KUKA KRL program: MsgLib.src, MsgLib.dat

--- MsgLib.src ---
&ACCESS RV1
&REL 15
&COMMENT Message library
DEF MsgLib()
   ;**************************************************
   ;Creation Date: 7.12.2007
   ;Change:  23.06.2012 additional properties possible
   ;         for logging and advance stop control
   ;Change:  16.06.2023 modify MsgNotifyTextPar
   ;Change:  06.09.2023 modify MsgNotifyTextPar & zip code
   ;**************************************************
   ;FOLD Interfaces and message examples within this fold
      ;----------Global subroutines and functions: -------
      ;MsgNotify(sText[]:IN, sModul[]:IN, nNumPar:IN, sTextPar[]:IN, nMsgNr:IN,MsgOpt:IN)
      ;MsgNotifyTextPar(sText[]:IN, sModul[]:IN, nNumPar:IN, sTextPar[]:IN, sTextPar2[]:IN, nMsgNr:IN,MsgOpt:IN)
      ;MsgQuit(sText[]:IN, sModul[]:IN, nNumPar:IN, sTextPar[]:IN, nMsgNr:IN,MsgOpt:IN)
      ;MsgState(nHandle:OUT, sText[]:IN, sModul[]:IN, nNumPar:IN, sTextPar[]:IN, nMsgNr:IN,MsgOpt:IN)
      ;MsgLoop(sText[]:IN,sModul[]:IN)
      ;MsgDialog(nAnswer:OUT,sText[]:IN,sModul[]:IN,sTextPar[]:IN,sDialogSK1[]:IN,sDialogSK2[]:IN,sDialogSK3[]:IN,sDialogSK4[]:IN,sDialogSK5[]:IN,sDialogSK6[]:IN,sDialogSK7[]:IN,NoBrakes:IN, nMsgNr:IN,MsgOpt:IN)
      ;----------Explainations for parameters: -----------
      ;CHAR sText[]  message text or message DB-key (80 chars)
      ;CHAR sModul[] (option) modulname or key (24 char)
      ;INT nNumPar   (option)numeric value inserted in sText[] at the position %1
      ;CHAR sTextPar[] (option)text or message DB-key inserted in sText[] at the position %1 (26 char)
      ;MsgOpt          (option) Structure KrlMsgOpt_T  BOOL VL_Stop,Clear_P_Reset,Log_To_DB
      ;                (option) VL_Stop=TRUE    => Creates an advance stop | FALSE avoids this behavior
      ;                (option) Clear_P_Reset=TRUE (Default) deletes Messages at program reset / cancelled
      ;                (option) Log_To_DB=TRUE => entry into logbook => enfluence to system performance
      ;----------Examples: -------------------------------
      ;MsgNotifyTextPar("Error", "CrossMeld", 0, "Error message 1", "Error message 2", 511)
      ;MsgNotify("this is a notify message")
      ;MsgQuit("this is a quit message", "myMod")
      ;MsgQuit("this is a quit message", "myMod",,,12345)
      ;INT myInt=123
      ;MsgQuit("this is the %1 quit message", "Module", myInt)
      ;MsgNotify("this is a %1 notify message", "Tech", , "asd")
      ;MsgLoop("this is the loop message")
      ;MsgLoop(" "); cancels loop message
      ;MsgDialog(DialogAnswer, "DBKEY" OR "dialog message", "Module", "TextPar for %1 in DBKey", "DialogKey1", "DialogKey2", "DialogKey3",,,,,,12345)
      ;MsgDialog(DialogAnswer, "StartPTP", "CrossMeld", "Achse 3", "YES", "NO", "Cancel")
      ;MsgNotifyTextPar("DBKEY" OR "notify message", "Module", 0 OR >0, "TextPar for %1", "TextPar for %2")
      ;  nNumPar = 0: TextPar will be send as %1 %2
      ;  nNumPar <> 0: nNumPar will be send as %1
      ;  nNumPar = ,,: TextPar will be send as %1 %2
   ;ENDFOLD
END


GLOBAL DEF MsgNotify(sText[]:IN, sModul[]:IN, nNumPar:IN, sTextPar[]:IN, nMsgNr:IN, MsgOpt:IN)
   DECL CHAR sText[]
   DECL CHAR sModul[]
   DECL CHAR sTextPar[]
   DECL KrlMsg_T Msg
   DECL KrlMsgParType_T MsgParType
   DECL KrlMsgPar_T MsgPar[3]
   DECL KrlMsgOpt_T MsgOpt ;Bool-elements: VL_Stop,Clear_P_Reset,Log_To_DB
   DECL KrlMsgOpt_T DummyMsgOpt
   DECL State_T State
   DECL INT count, len, offset, nHandle
   DECL INT nNumPar
   DECL INT nMsgNr
   CheckOfMsgOpt(MsgOpt);Creates default values in case of none availability
   CheckOfMsgNr(Msg, nMsgNr);Creates default values in case of none availability
   CheckOfMsgText(Msg, sText[])
   CheckOfModulText(Msg, sModul[])
   ERR_CLEAR($ERR)
   ON_ERROR_PROCEED
   offset=nNumPar
   IF $ERR.Number == 0 THEN
      offset=0
      MsgPar[1].Par_Txt[]=" "
      Swrite(MsgPar[1].Par_Txt[], State, Offset, "%d", nNumPar)
      MsgPar[1].Par_type=#Value
   ELSE
      ERR_CLEAR($ERR)
      ON_ERROR_PROCEED
      len=STRLEN(sTextPar[])
      IF len > 0 THEN
         IF len > 26 THEN
            len=26
         ENDIF
         FOR count = 1 TO len
            MsgPar[1].Par_Txt[count]=sTextPar[count]
         ENDFOR
         MsgPar[1].Par_type=#Value
      ENDIF
   ENDIF
   nHandle=Set_KrlMsg(#NOTIFY, Msg, MsgPar[], MsgOpt)
END


GLOBAL DEF MsgQuit(sText[]:IN, sModul[]:IN, nNumPar:IN, sTextPar[]:IN, nMsgNr:IN, MsgOpt:IN)
   DECL CHAR sText[]
   DECL CHAR sModul[]
   DECL CHAR sTextPar[]
   DECL KrlMsg_T Msg
   DECL KrlMsgParType_T MsgParType
   DECL KrlMsgPar_T MsgPar[3]
   DECL KrlMsgOpt_T MsgOpt
   DECL KrlMsgOpt_T DummyMsgOpt
   DECL State_T State
   DECL INT count, len, offset, nHandle
   DECL INT nNumPar
   DECL INT nMsgNr
   CheckOfMsgOpt(MsgOpt);Creates default values in case of none availability
   CheckOfMsgNr(Msg, nMsgNr);Creates default values in case of none availability
   CheckOfMsgText(Msg, sText[])
   CheckOfModulText(Msg, sModul[])
   ERR_CLEAR($ERR)
   ON_ERROR_PROCEED
   offset=nNumPar
   IF $ERR.Number == 0 THEN
      offset=0
      MsgPar[1].Par_Txt[]=" "
      Swrite(MsgPar[1].Par_Txt[], State, offset, "%d", nNumPar)
      MsgPar[1].Par_type=#Value
   ELSE
      ERR_CLEAR($ERR)
      len=STRLEN(sTextPar[])
      IF len > 0 THEN
         IF len > 26 THEN
            len=26
         ENDIF
         FOR count = 1 TO len
            MsgPar[1].Par_Txt[count]=sTextPar[count]
         ENDFOR
         MsgPar[1].Par_type=#Value
      ENDIF
   ENDIF
   nHandle=Set_KrlMsg(#QUIT, Msg, MsgPar[], MsgOpt)
   WHILE (Exists_KrlMsg(nHandle))
      WAIT SEC 0.1
   ENDWHILE
END


GLOBAL DEF MsgState(nHandle:OUT, sText[]:IN, sModul[]:IN, nNumPar:IN, sTextPar[]:IN, nMsgNr:IN, MsgOpt:IN)
   DECL CHAR sText[]
   DECL CHAR sModul[]
   DECL CHAR sTextPar[]
   DECL KrlMsg_T Msg
   DECL KrlMsgParType_T MsgParType
   DECL KrlMsgPar_T MsgPar[3]
   DECL KrlMsgOpt_T MsgOpt
   DECL KrlMsgOpt_T DummyMsgOpt
   DECL State_T State
   DECL INT count, len, offset
   DECL INT nHandle
   DECL INT nNumPar
   DECL INT nMsgNr
   CheckOfMsgOpt(MsgOpt);Creates default values in case of none availability
   CheckOfMsgNr(Msg, nMsgNr);Creates default values in case of none availability
   CheckOfMsgText(Msg, sText[])
   CheckOfModulText(Msg, sModul[])
   ERR_CLEAR($ERR)
   ON_ERROR_PROCEED
   offset=nNumPar
   IF $ERR.Number == 0 THEN
      offset=0
      MsgPar[1].Par_Txt[]=" "
      Swrite(MsgPar[1].Par_Txt[], State, offset, "%d", nNumPar)
      MsgPar[1].Par_type=#Value
   ELSE
      ERR_CLEAR($ERR)
      len=STRLEN(sTextPar[])
      IF len > 0 THEN
         IF len > 26 THEN
            len=26
         ENDIF
         FOR count = 1 TO len
            MsgPar[1].Par_Txt[count]=sTextPar[count]
         ENDFOR
         MsgPar[1].Par_type=#Value
      ENDIF
   ENDIF
   nHandle=Set_KrlMsg(#STATE, Msg, MsgPar[], MsgOpt)
END


GLOBAL DEF MsgLoop(sText[]:IN, sModul[]:IN)
   DECL CHAR sText[]
   DECL CHAR sModul[]
   DECL CHAR sMsg[80]
   DECL CHAR sMod[24]
   DECL INT count, len
   len=STRLEN(sText[])
   IF len > 0 THEN
      IF len > 80 THEN
         len=80
      ENDIF
      FOR count = 1 TO len
         sMsg[count]=sText[count]
      ENDFOR
   ENDIF
   len=STRLEN(sModul[])
   IF len > 0 THEN
      IF len > 24 THEN
         len=24
      ENDIF
      FOR count = 1 TO len
         sMod[count]=sModul[count]
      ENDFOR
   ELSE
      sMod[]="Appl"
   ENDIF
   IF (STRLEN(sMsg[]) > 0) THEN
      IF lnHandle > 0 THEN
         WAIT FOR Clear_KrlMsg(lnHandle) OR TRUE
         lnHandle=0
      ENDIF
      FOR count = 1 TO STRLEN(sMsg[])
         IF sMsg[count] <> " " THEN
            MsgState(lnHandle, sMsg[], sMod[])
            EXIT
         ENDIF
      ENDFOR
   ENDIF
END


GLOBAL DEF MsgDialog(nAnswer:OUT, sText[]:IN, sModul[]:IN, sTextPar[]:IN, sDialogSK1[]:IN, sDialogSK2[]:IN, sDialogSK3[]:IN, sDialogSK4[]:IN, sDialogSK5[]:IN, sDialogSK6[]:IN, sDialogSK7[]:IN, NoBrakes:IN, nMsgNr:IN, MsgOpt:IN)
   DECL KrlMsg_T Msg
   DECL KrlMsgPar_T MsgPar[3]
   DECL KrlMsgOpt_T MsgOpt
   DECL KrlMsgOpt_T DummyMsgOpt
   DECL KrlMsgDlgSK_T Msg_SOFTKEY[7]
   DECL INT count, len, nHandle
   DECL INT nAnswer
   DECL INT nMsgNr
   DECL BOOL NoBrakes
   DECL CHAR sText[]
   DECL CHAR sModul[]
   DECL CHAR sTextPar[]
   DECL CHAR sDialogSK1[]
   DECL CHAR sDialogSK2[]
   DECL CHAR sDialogSK3[]
   DECL CHAR sDialogSK4[]
   DECL CHAR sDialogSK5[]
   DECL CHAR sDialogSK6[]
   DECL CHAR sDialogSK7[]
   DECL CHAR sMsg[80]
   CheckOfMsgOpt(MsgOpt);Creates default values in case of none availability
   CheckOfMsgNr(Msg, nMsgNr);Creates default values in case of none availability
   CheckOfMsgText(Msg, sText[])
   CheckOfModulText(Msg, sModul[])
   ERR_CLEAR($ERR)
   ON_ERROR_PROCEED
   len=STRLEN(sDialogSK1[])
   IF $ERR.Number == 0 THEN
      IF len > 0 THEN
         IF len > 24 THEN
            len=24
         ENDIF
         Msg_SOFTKEY[7].Sk_Type=#KEY
         FOR count = 1 TO len
            Msg_SOFTKEY[7].Sk_txt[count]=sDialogSK1[count]
         ENDFOR
      ENDIF
   ELSE
      FOR count = 1 TO 24
         Msg_SOFTKEY[7].Sk_txt[count]=" "
      ENDFOR
   ENDIF
   ERR_CLEAR($ERR)
   ON_ERROR_PROCEED
   len=STRLEN(sDialogSK2[])
   IF $ERR.Number == 0 THEN
      len=STRLEN(sDialogSK2[])
      IF len > 0 THEN
         IF len > 24 THEN
            len=24
         ENDIF
         Msg_SOFTKEY[6].Sk_Type=#KEY
         FOR count = 1 TO len
            Msg_SOFTKEY[6].Sk_txt[count]=sDialogSK2[count]
         ENDFOR
      ENDIF
   ELSE
      FOR count = 1 TO 24
         Msg_SOFTKEY[6].Sk_txt[count]=" "
      ENDFOR
   ENDIF
   ERR_CLEAR($ERR)
   ON_ERROR_PROCEED
   len=STRLEN(sDialogSK3[])
   IF $ERR.Number == 0 THEN
      len=STRLEN(sDialogSK3[])
      IF len > 0 THEN
         IF len > 24 THEN
            len=24
         ENDIF
         Msg_SOFTKEY[5].Sk_Type=#KEY
         FOR count = 1 TO len
            Msg_SOFTKEY[5].Sk_txt[count]=sDialogSK3[count]
         ENDFOR
      ENDIF
   ELSE
      FOR count = 1 TO 24
         Msg_SOFTKEY[5].Sk_txt[count]=" "
      ENDFOR
   ENDIF
   ERR_CLEAR($ERR)
   ON_ERROR_PROCEED
   len=STRLEN(sDialogSK4[])
   IF $ERR.Number == 0 THEN
      len=STRLEN(sDialogSK4[])
      IF len > 0 THEN
         IF len > 24 THEN
            len=24
         ENDIF
         Msg_SOFTKEY[4].Sk_Type=#KEY
         FOR count = 1 TO len
            Msg_SOFTKEY[4].Sk_txt[count]=sDialogSK4[count]
         ENDFOR
      ENDIF
   ELSE
      FOR count = 1 TO 24
         Msg_SOFTKEY[4].Sk_txt[count]=" "
      ENDFOR
   ENDIF
   ERR_CLEAR($ERR)
   ON_ERROR_PROCEED
   len=STRLEN(sDialogSK5[])
   IF $ERR.Number == 0 THEN
      len=STRLEN(sDialogSK5[])
      IF len > 0 THEN
         IF len > 24 THEN
            len=24
         ENDIF
         Msg_SOFTKEY[3].Sk_Type=#KEY
         FOR count = 1 TO len
            Msg_SOFTKEY[3].Sk_txt[count]=sDialogSK5[count]
         ENDFOR
      ENDIF
   ELSE
      FOR count = 1 TO 24
         Msg_SOFTKEY[3].Sk_txt[count]=" "
      ENDFOR
   ENDIF
   ERR_CLEAR($ERR)
   ON_ERROR_PROCEED
   len=STRLEN(sDialogSK6[])
   IF $ERR.Number == 0 THEN
      len=STRLEN(sDialogSK6[])
      IF len > 0 THEN
         IF len > 24 THEN
            len=24
         ENDIF
         Msg_SOFTKEY[2].Sk_Type=#KEY
         FOR count = 1 TO len
            Msg_SOFTKEY[2].Sk_txt[count]=sDialogSK6[count]
         ENDFOR
      ENDIF
   ELSE
      FOR count = 1 TO 24
         Msg_SOFTKEY[2].Sk_txt[count]=" "
      ENDFOR
   ENDIF
   ERR_CLEAR($ERR)
   ON_ERROR_PROCEED
   len=STRLEN(sDialogSK7[])
   IF $ERR.Number == 0 THEN
      len=STRLEN(sDialogSK7[])
      IF len > 0 THEN
         IF len > 24 THEN
            len=24
         ENDIF
         Msg_SOFTKEY[1].Sk_Type=#KEY
         FOR count = 1 TO len
            Msg_SOFTKEY[1].Sk_txt[count]=sDialogSK7[count]
         ENDFOR
      ENDIF
   ELSE
      FOR count = 1 TO 24
         Msg_SOFTKEY[1].Sk_txt[count]=" "
      ENDFOR
   ENDIF
   len=STRLEN(sTextPar[])
   IF len > 0 THEN
      IF len > 26 THEN
         len=26
      ENDIF
      FOR count = 1 TO len
         MsgPar[1].Par_Txt[count]=sTextPar[count]
      ENDFOR
      MsgPar[1].Par_type=#Value
   ENDIF
   nHandle=SET_KRLDLG(Msg, MsgPar[], Msg_SOFTKEY[], MsgOpt)
   ERR_CLEAR($ERR)
   ON_ERROR_PROCEED
   NoBrakes=NoBrakes
   IF NOT ($ERR.Number == 0) THEN
      NoBrakes=FALSE
   ENDIF
   IF (nHandle > 0) THEN
      WHILE (Exists_KrlDlg(nHandle, nAnswer))
         WAIT SEC 0.5
         IF NoBrakes THEN
            PTP $AXIS_ACT
         ENDIF
      ENDWHILE
   ENDIF
END


GLOBAL DEF MsgNotifyTextPar(sText[]:IN, sModul[]:IN, nNumPar:IN, sTextPar[]:IN, sTextPar2[]:IN, nMsgNr:IN, MsgOpt:IN)
   DECL CHAR sText[]
   DECL CHAR sModul[]
   DECL CHAR sTextPar[]
   DECL CHAR sTextPar2[]
   DECL KrlMsg_T Msg
   DECL EKrlMsgType MsgType
   DECL KrlMsgParType_T MsgParType
   DECL KrlMsgPar_T MsgPar[3]
   DECL KrlMsgOpt_T MsgOpt
   DECL KrlMsgOpt_T DummyMsgOpt
   DECL State_T State
   DECL INT count, len, offset, nHandle
   DECL INT nNumPar
   DECL INT nMsgNr
   MsgType=#Notify
   CheckOfMsgOpt(MsgOpt);Creates default values in case of none availability
   CheckOfMsgNr(Msg, nMsgNr);Creates default values in case of none availability
   CheckOfMsgText(Msg, sText[])
   CheckOfModulText(Msg, sModul[])
   ON_ERROR_PROCEED
   offset=nNumPar
   IF ($ERR.Number <> 0) THEN
      nNumPar=0 ;If no int parameter is given set value to 0. TextPar will be send as %1 %2
      ERR_CLEAR($ERR)
   ENDIF
   IF nNumPar == 0 THEN
      ; 1st Parameter
      len=STRLEN(sTextPar[])
      IF len > 0 THEN
         IF len > 26 THEN
            len=26
         ENDIF
         FOR count = 1 TO len
            MsgPar[1].Par_Txt[count]=sTextPar[count]
         ENDFOR
         MsgPar[1].Par_type=#Value
      ELSE
         MsgPar[1].Par_Txt[]=" "
         MsgPar[1].Par_type=#Value
      ENDIF
      ; 2nd Parameter
      len=STRLEN(sTextPar2[])
      IF len > 0 THEN
         IF len > 26 THEN
            len=26
         ENDIF
         FOR count = 1 TO len
            MsgPar[2].Par_Txt[count]=sTextPar2[count]
         ENDFOR
         MsgPar[2].Par_type=#Value
      ELSE
         MsgPar[2].Par_Txt[]=" "
         MsgPar[2].Par_type=#Value
      ENDIF
   ELSE
      offset=0
      MsgPar[1].Par_Txt[]=" "
      Swrite(MsgPar[1].Par_Txt[], State, Offset, "%d", nNumPar)
      MsgPar[1].Par_type=#Value
      MsgPar[2].Par_Txt[]=" "
      MsgPar[2].Par_type=#Value
   ENDIF
   nHandle=Set_KrlMsg(MsgType, Msg, MsgPar[], MsgOpt)
END


GLOBAL DEF MsgQuitTextPar(sText[]:IN, sModul[]:IN, nNumPar:IN, sTextPar[]:IN, sTextPar2[]:IN, nMsgNr:IN, MsgOpt:IN)
   DECL CHAR sText[]
   DECL CHAR sModul[]
   DECL CHAR sTextPar[]
   DECL CHAR sTextPar2[]
   DECL KrlMsg_T Msg
   DECL EKrlMsgType MsgType
   DECL KrlMsgParType_T MsgParType
   DECL KrlMsgPar_T MsgPar[3]
   DECL KrlMsgOpt_T MsgOpt
   DECL KrlMsgOpt_T DummyMsgOpt
   DECL State_T State
   DECL INT count, len, offset, nHandle
   DECL INT nNumPar
   DECL INT nMsgNr
   MsgType=#QUIT
   CheckOfMsgOpt(MsgOpt);Creates default values in case of none availability
   CheckOfMsgNr(Msg, nMsgNr);Creates default values in case of none availability
   CheckOfMsgText(Msg, sText[])
   CheckOfModulText(Msg, sModul[])
   ON_ERROR_PROCEED
   offset=nNumPar
   IF ($ERR.Number <> 0) THEN
      nNumPar=0 ;If no int parameter is given set value to 0. TextPar will be send as %1 %2
      ERR_CLEAR($ERR)
   ENDIF
   IF nNumPar == 0 THEN
      ; 1st Parameter
      len=STRLEN(sTextPar[])
      IF len > 0 THEN
         IF len > 26 THEN
            len=26
         ENDIF
         FOR count = 1 TO len
            MsgPar[1].Par_Txt[count]=sTextPar[count]
         ENDFOR
         MsgPar[1].Par_type=#Value
      ELSE
         MsgPar[1].Par_Txt[]=" "
         MsgPar[1].Par_type=#Value
      ENDIF
      ; 2nd Parameter
      len=STRLEN(sTextPar2[])
      IF len > 0 THEN
         IF len > 26 THEN
            len=26
         ENDIF
         FOR count = 1 TO len
            MsgPar[2].Par_Txt[count]=sTextPar2[count]
         ENDFOR
         MsgPar[2].Par_type=#Value
      ELSE
         MsgPar[2].Par_Txt[]=" "
         MsgPar[2].Par_type=#Value
      ENDIF
   ELSE
      offset=0
      MsgPar[1].Par_Txt[]=" "
      Swrite(MsgPar[1].Par_Txt[], State, Offset, "%d", nNumPar)
      MsgPar[1].Par_type=#Value
      MsgPar[2].Par_Txt[]=" "
      MsgPar[2].Par_type=#Value
   ENDIF
   nHandle=Set_KrlMsg(MsgType, Msg, MsgPar[], MsgOpt)
END


DEF CheckOfMsgOpt(LocalMsgOpt:OUT)
   DECL KrlMsgOpt_T LocalMsgOpt ;Bool-elements: VL_Stop,Clear_P_Reset,Log_To_DB
   DECL KrlMsgOpt_T DummyMsgOpt
   ;Default Values: MsgOpt={ VL_Stop TRUE, Clear_P_Reset TRUE, Log_To_DB False }
   ON_ERROR_PROCEED
   DummyMsgOpt.VL_Stop=LocalMsgOpt.VL_Stop
   IF ($ERR.Number <> 0) THEN
      LocalMsgOpt.VL_Stop=TRUE ;DEFAULT setting TRUE
      ERR_CLEAR($ERR)
   ENDIF
   ON_ERROR_PROCEED
   DummyMsgOpt.Clear_P_Reset=LocalMsgOpt.Clear_P_Reset
   IF ($ERR.Number <> 0) THEN
      LocalMsgOpt.Clear_P_Reset=TRUE ;DEFAULT setting TRUE
      ERR_CLEAR($ERR)
   ENDIF
   ON_ERROR_PROCEED
   DummyMsgOpt.Log_To_DB=LocalMsgOpt.Log_To_DB
   IF ($ERR.Number <> 0) THEN
      LocalMsgOpt.Log_To_DB=FALSE ;DEFAULT setting FALSE
      ERR_CLEAR($ERR)
   ENDIF
END


DEF CheckOfMsgNr(LocalMsg:OUT, LocalMsgNr:OUT)
   DECL INT LocalMsgNr
   DECL KrlMsg_T LocalMsg
   ;Default Values: Msg.Nr=1
   ON_ERROR_PROCEED
   LocalMsg.Nr=LocalMsgNr
   IF ($ERR.Number <> 0) THEN
      LocalMsg.Nr=1
      ERR_CLEAR($ERR)
   ENDIF
END


DEF CheckOfMsgText(LocalMsg:OUT, LocalText[]:OUT)
   DECL CHAR LocalText[]
   DECL KrlMsg_T LocalMsg
   DECL INT len, count
   len=STRLEN(LocalText[])
   IF len > 0 THEN
      IF len > 80 THEN
         len=80
      ENDIF
      FOR count = 1 TO len
         LocalMsg.Msg_txt[count]=LocalText[count]
      ENDFOR
   ELSE
      LocalMsg.Msg_txt[]="parameter sText[] is missing"
   ENDIF
END


DEF CheckOfModulText(LocalMsg:OUT, LocalModul[]:OUT)
   DECL CHAR LocalModul[]
   DECL KrlMsg_T LocalMsg
   DECL INT len, count
   len=STRLEN(LocalModul[])
   IF len > 0 THEN
      IF len > 24 THEN
         len=24
      ENDIF
      FOR count = 1 TO len
         LocalMsg.Modul[count]=LocalModul[count]
      ENDFOR
   ELSE
      LocalMsg.Modul[]="Appl"
   ENDIF
END

--- MsgLib.dat ---
&ACCESS  R
&COMMENT Message library
DEFDAT  MsgLib PUBLIC

   DECL INT lnHandle=0

ENDDAT
